PROGRAM PRG_TEST
VAR
	Drive_Test	: FB_DRIVE_TEST;
END_VAR

TcUnit.RUN();

END_PROGRAM

(* stored: Version 1.1.0.1, ProductVersion 3.1.4024.12
   POU PRG_TEST: Id {b211fc4f-8cea-4f4f-a425-ec32459017bc}, SpecialFunc None *)
